{attribute 'linkalways'} 
{attribute 'no_explicit_call' := 'This FB is a CLASS and must be accessed using methods or properties'}
{attribute 'enable_dynamic_creation'}
FUNCTION_BLOCK CreateGraphMultiUserRpcHandler IMPLEMENTS I_AsynchronousRpcHandler
VAR
	graphFramework : I_GraphFramework;
	graphs : I_Graphs;
	userGraphs : Dictionary;
END_VAR

METHOD Handle
VAR_INPUT
	Parameters : I_Deserializer;
	Response : I_AsynchronousRpcResponse;
END_VAR
VAR
	clientId : T_MAXSTRING;
	graphUuid : T_MAXSTRING;
	graph : I_Graph;
	feedback : DeserializerFeedback;
	graphDeserializer : I_Deserializer;
	serializer : I_Serializer;
	getStatusVisitor : GetStatusVisitor;
END_VAR
IF NOT Parameters.TryGetKeyString('clienId', clientId, feedback) THEN
	Response.RejectWithMessage(feedback.FirstError.Message);
	RETURN;
END_IF

IF NOT userGraphs.TryGetValue(clientId, graphUuid) THEN
	IF graphs.TryGetGraphByUuid(graphUuid,graph) THEN
		graphs.RemoveGraph(graph);
		graph.Dispose();
	END_IF
	userGraphs.Remove(clientId);
END_IF

graph := graphFramework.Create();
graphDeserializer := Parameters.GetKeyObject('graph');

IF NOT graph.TryDeserializeFrom(graphDeserializer, feedback) THEN
	Response.RejectWithMessage(feedback.FirstError.Message);
	graph.Dispose();
	RETURN;
END_IF

graphUuid := graph.Uuid;
userGraphs.AddOrUpdate(clientId, graphUuid);
graphs.AddGraph(graph);

serializer := Response.GetSerializer();
getStatusVisitor.Initialize(serializer);
getStatusVisitor.VisitGraph(graph);
Response.CompleteWithSerializer(serializer);
serializer.Dispose();
END_METHOD

METHOD PUBLIC Initialize
VAR_INPUT
	GraphFramework : I_GraphFramework;
	Graphs : I_Graphs;
END_VAR
THIS^.graphFramework := GraphFramework;
THIS^.graphs := Graphs;
END_METHOD

END_FUNCTION_BLOCK

(* stored: Version 1.1.0.1, ProductVersion 3.1.4024.12
   POU CreateGraphMultiUserRpcHandler: Id {d6b88ddc-1f3f-4bc6-9cec-7511e5f75694}, SpecialFunc None
   Method Handle: Id {2fa8f613-f7ff-45a2-bdd0-f1d9eaa294a4}
   Method Initialize: Id {6117f436-a2fa-4784-a767-69b747ee1b47} *)
